// TIA Portal V20 export
DATA_BLOCK "SyncNode"   // DB21
{ DB_Accessible_From_OPC_UA := 'FALSE' }
// stored: DBAccessibleFromOPCUA false, DBAccessibleFromWebserver false, InstanceOfName Unit1.Em0.typeSyncNode, InstanceOfType UDT, Namespace Unit1.Em0
"Unit1.Em0.typeSyncNode"
   // VAR
   //    commands { ExternalWritable := 'False'} : Struct
   //       enableHpMotion : Bool := FALSE;
   //    END_STRUCT;
   //    status { ExternalWritable := 'False'} : Struct
   //       busy : Bool := FALSE;
   //       error : Bool := FALSE;
   //    END_STRUCT;
   //    WinderInput { S7_SetPoint := 'True'} : "LConSMC_typeWinderInput";
   //    WinderOutput { S7_SetPoint := 'True'} : "LConSMC_typeWinderOutput";
   //    WinderConfig { S7_SetPoint := 'True'} : "LConSMC_typeWinderConfig";
   //    WinderDiag { S7_SetPoint := 'True'} : "LConSMC_typeWinderDiag";
   // END_VAR
BEGIN
   WinderInput.enable := FALSE;
   WinderInput.speedMatch := FALSE;
   WinderInput.cntrlEnable := FALSE;
   WinderInput.jogPos := FALSE;
   WinderInput.jogNeg := FALSE;
   WinderInput.lineAxisMotionVector.s := 0.0;
   WinderInput.lineAxisMotionVector.v := 0.0;
   WinderInput.lineAxisMotionVector."a" := 0.0;
   WinderInput.lineAxisActualValues.s := 0.0;
   WinderInput.lineAxisActualValues.v := 0.0;
   WinderInput.additionalVelocity := 0.0;
   WinderInput.typeOfWinder := 2;
   WinderInput.controlMode := 0;
   WinderInput.typeOfDiameterCalc := 3;
   WinderInput.holdDiameter := FALSE;
   WinderInput.setDiameter := FALSE;
   WinderInput.CntrlSetpoint := 0.0;
   WinderInput.CntrlActual := 24.9056603773585;
   WinderInput.tCycle := 2.0;
   WinderInput.winderAxis := 263;
   WinderOutput.busy := FALSE;
   WinderOutput.active := FALSE;
   WinderOutput.ctrlBusy := FALSE;
   WinderOutput.inSync := FALSE;
   WinderOutput.error := FALSE;
   WinderOutput.errorID := 16#0000_0000;
   WinderConfig.positionControlled := FALSE;
   WinderConfig.axisCtrl := TRUE;
   WinderConfig.jogVelocity := 10.0;
   WinderConfig.overrideVelocity := 0.0;
   WinderConfig.maxVelocity := 100.0;
   WinderConfig.getAxisConfigAtStart := TRUE;
   WinderConfig.noOfSamplesLineVelocity := 1;
   WinderConfig.unitConfiguration.metricUnits := TRUE;
   WinderConfig.unitConfiguration.axisVelocityUnit := 1521;
   WinderConfig.unitConfiguration.axisTorqueUnit := 1126;
   WinderConfig.winderDynamics.stopDynamics.deceleration := 360.0;
   WinderConfig.winderDynamics.stopDynamics.jerk := 0.0;
   WinderConfig.winderDynamics.stopDynamics.abortAcceleration := TRUE;
   WinderConfig.winderDynamics.syncDynamics.acceleration := 360.0;
   WinderConfig.winderDynamics.syncDynamics.deceleration := 360.0;
   WinderConfig.winderDynamics.syncDynamics.jerk := 0.0;
   WinderConfig.winderDynamics.syncDynamics.abortAcceleration := FALSE;
   WinderConfig.winderDynamics.syncDynamics.syncToleranceFactor := 1.0;
   WinderConfig.winderDynamics.operationDynamics.acceleration := 360000.0;
   WinderConfig.winderDynamics.operationDynamics.deceleration := 360000.0;
   WinderConfig.winderDynamics.operationDynamics.jerk := 0.0;
   WinderConfig.winderDynamics.jogDynamics.acceleration := 360.0;
   WinderConfig.winderDynamics.jogDynamics.deceleration := 360.0;
   WinderConfig.winderDynamics.jogDynamics.jerk := 0.0;
   WinderConfig.torquePrecontrolConfig.useSetValForFrictionComp := TRUE;
   WinderConfig.torquePrecontrolConfig.frictionAdjustment := 0.0;
   WinderConfig.torquePrecontrolConfig.xn_speedValues.values[0..19] := 0.0;
   WinderConfig.torquePrecontrolConfig.yn_torqueValues.values[0..19] := 0.0;
   WinderConfig.torquePrecontrolConfig.sizeOfArray := 20;
   WinderConfig.torquePrecontrolConfig.loadGear.numerator := 30;
   WinderConfig.torquePrecontrolConfig.loadGear.denominator := 1;
   WinderConfig.torquePrecontrolConfig.MaterialWidth := 0.035;
   WinderConfig.torquePrecontrolConfig.MaterialDensity := 2700.0;
   WinderConfig.torquePrecontrolConfig.MaterialFillFactor := 1.0;
   WinderConfig.torquePrecontrolConfig.JFixed := 0.0327900014817715;
   WinderConfig.torquePrecontrolConfig.JMandrel := 0.1;
   WinderConfig.torquePrecontrolConfig.JMotor := 0.00104;
   WinderConfig.torquePrecontrolConfig.tensionAdjustment := 0.5;
   WinderConfig.torquePrecontrolConfig.accelerationAdjustment := 0.1;
   WinderConfig.torquePrecontrolConfig.dDdTAdjustment := 0.0;
   WinderConfig.torquePrecontrolConfig.upperTorqueLimit := 0.2;
   WinderConfig.torquePrecontrolConfig.lowerTorqueLimit := -0.2;
   WinderConfig.torquePrecontrolConfig.referenceTorque := 11.55;
   WinderConfig.torquePrecontrolConfig.additiveTorque := 0.0;
   WinderConfig.diamConfig.minLineVelocity := 0.5;
   WinderConfig.diamConfig.minShaftSpeed := 0.0;
   WinderConfig.diamConfig.minDia := 0.08;
   WinderConfig.diamConfig.maxDia := 0.4;
   WinderConfig.diamConfig.webThickness := 0.0001275;
   WinderConfig.diamConfig.useLineAxisActualValues := TRUE;
   WinderConfig.diamConfig.diameterSetValue := 0.1876;
   WinderConfig.diamConfig.lineFilterTime := 20.0;
   WinderConfig.diamConfig.shaftFilterTime := 20.0;
   WinderConfig.diamConfig.measuringRevolutionCount := 4.0;
   WinderConfig.diamConfig.firstDiameterOutput := 0.5;
   WinderConfig.diamConfig.diameterOutputRate := 1.0;
   WinderConfig.diamConfig.lineModLength := 1.0;
   WinderConfig.diamConfig.shaftModLength := 360.0;
   WinderConfig.diamConfig.diameterFilterTime := 360.0;
   WinderConfig.technologyControllerConfig.x1 := 0.0;
   WinderConfig.technologyControllerConfig.Kp1 := 3.0;
   WinderConfig.technologyControllerConfig.x2 := 0.0;
   WinderConfig.technologyControllerConfig.Kp2 := 0.0;
   WinderConfig.technologyControllerConfig.KpAdaptionValue := 0.0;
   WinderConfig.technologyControllerConfig.integTime := 2000.0;
   WinderConfig.technologyControllerConfig.derivTime := 0.0;
   WinderConfig.technologyControllerConfig.derivControlMode := FALSE;
   WinderConfig.technologyControllerConfig.setNominalValue := 100.0;
   WinderConfig.technologyControllerConfig.setRampTime := 10000.0;
   WinderConfig.technologyControllerConfig.filterTime := 10.0;
   WinderConfig.technologyControllerConfig.intSetValue := 0.0;
   WinderConfig.technologyControllerConfig.setIntChannel := FALSE;
   WinderConfig.technologyControllerConfig.holdIntChannel := FALSE;
   WinderConfig.technologyControllerConfig.deadBand := 0.0;
   WinderConfig.technologyControllerConfig.outValueFactor := 1.0;
   WinderConfig.technologyControllerConfig.upperLimit := 2.0;
   WinderConfig.technologyControllerConfig.lowerLimit := -2.0;
   WinderConfig.technologyControllerConfig.limRampTime := 300.0;
   WinderConfig.technologyControllerConfig.tensionReference := 0.0;
   WinderConfig.webbreakDetectionConfig.enableDetection := FALSE;
   WinderConfig.webbreakDetectionConfig.minLineVelocity := 5.0;
   WinderConfig.webbreakDetectionConfig.upperLimitError := 0.5;
   WinderConfig.webbreakDetectionConfig.lowerLimitError := 0.5;
   WinderConfig.webbreakDetectionConfig.delayTime := T#200MS;
   WinderDiag.typeOfAxis := 0;
   WinderDiag.referenceVelocity := 0.0;
   WinderDiag.diameterFactor := 0.0;
   WinderDiag.diamCalcDiag.atMinDia := FALSE;
   WinderDiag.diamCalcDiag.atMaxDia := FALSE;
   WinderDiag.diamCalcDiag.diamIsHold := FALSE;
   WinderDiag.diamCalcDiag.calculatedWebThickness := 0.0;
   WinderDiag.torquePreControlDiag.upperTorqueLimit := 0.0;
   WinderDiag.torquePreControlDiag.lowerTorqueLimit := 0.0;
   WinderDiag.torquePreControlDiag.totalTorquePreControl := 0.0;
   WinderDiag.torquePreControlDiag.totalInertia := 0.0;
   WinderDiag.torquePreControlDiag.maxInertia := 0.0;
   WinderDiag.torquePreControlDiag.referenceTorque := 0.0;
   WinderDiag.torquePreControlDiag.loadGear.numerator := 1;
   WinderDiag.torquePreControlDiag.loadGear.denominator := 1;
   WinderDiag.technologyControllerDiag.pidoutValue := 0.0;
   WinderDiag.technologyControllerDiag.pidEffectiveKp := 0.0;
   WinderDiag.technologyControllerDiag.pidUpperLimitReached := FALSE;
   WinderDiag.technologyControllerDiag.pidLowerLimitReached := FALSE;
   WinderDiag.technologyControllerDiag.pidRFGSetpointReached := FALSE;
   WinderDiag.webbreakDiag.webbreakDetectionActive := FALSE;
   WinderDiag.webbreakDiag.webBreak := FALSE;
END_DATA_BLOCK
